TYPE ST_PopUp_FromHmi :
STRUCT
	stButton01	: ST_HMI_BUTTON_IN;
	stButton02	: ST_HMI_BUTTON_IN;
	stButton03	: ST_HMI_BUTTON_IN;
	stButton04	: ST_HMI_BUTTON_IN;
END_STRUCT
END_TYPE

(* stored: Version 1.1.0.1, ProductVersion 3.1.4024.11
   DUT ST_PopUp_FromHmi: Id {50925b52-00cf-4cde-a52f-11f6b01f98a9} *)
